// LS Electric XG5000 project: 8_22_2
// PLC LSPLC

PROGRAM NewProgram (task: 스캔 프로그램)

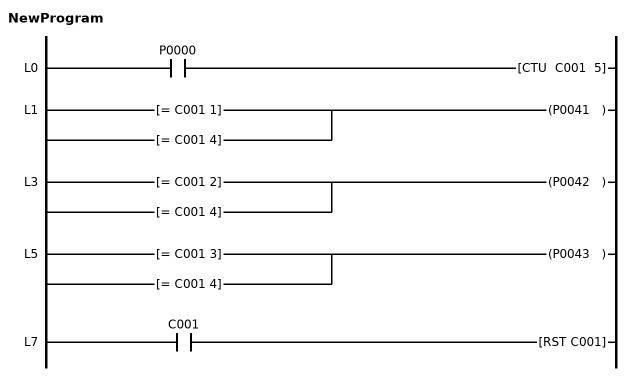
; L0
LOAD      P0000
CTU       C001 5
; L1
LOAD=     C001 1
OR=       C001 4
OUT       P0041
; L3
LOAD=     C001 2
OR=       C001 4
OUT       P0042
; L5
LOAD=     C001 3
OR=       C001 4
OUT       P0043
; L7
LOAD      C001
RST       C001